// TIA Portal project "Phanloai_SP_height" (V16)
// Vorlageprojekt für das Buch mit Zielsystem S7-1200

(* hardware
DEVICE "S7-1200-Station_1"  S7-1200 Station
   slot 0: "Baugruppenträger_0"  Rack  V1.0
   slot 1: "PLC_1"  CPU 1211C DC/DC/DC  6ES7 211-1AE40-0XB0  V4.1
DEVICE "PC-System_1"  SIMATIC PC station
   slot 0: "SIMATIC PC station"  Rail  SIMATIC PC-Station  V1.0
      slot 125: "Stationmanager"  Station_Manager  V6.0.4
   slot 1: "HMI_RT_1"  WinCC RT Advanced  6AV2 104-0xxxx-xxxx  16.0.0.0
      slot 33792: "Computer interface"  Host interface
   slot 2: "IE general_1"  IE General  IE_CP  V8.2.0
*)

// ===== PLC "PLC_1"  CPU 1211C DC/DC/DC =====

VAR_GLOBAL   // PLC tag table "Standard-Variablentabelle"
   "M_Start" AT %M10.0 : Bool;
   "M_Stop" AT %M10.1 : Bool;
   "Den_M_Start" AT %M10.5 : Bool;
   "M_Pause" AT %M10.2 : Bool;
END_VAR

VAR_GLOBAL   // PLC tag table "INOUT"
   "START" AT %E0.0 : Bool;
   "STOP" AT %E0.1 : Bool;
   "Den START" AT %Q0.5 : Bool;
   "BT1" AT %A0.0 : Bool;
   "SS0" AT %I0.2 : Bool;
   "Pusher 0" AT %Q0.1 : Bool;
   "BT2" AT %Q0.4 : Bool;
   "PAUSE" AT %I0.5 : Bool;
   "SS1" AT %I0.3 : Bool;
   "Pusher 1" AT %Q0.2 : Bool;
   "Light 0" AT %Q1.0 : Bool;
   "Light 1" AT %Q1.1 : Bool;
   "Light 2" AT %Q1.2 : Bool;
   "Den STOP" AT %Q0.7 : Bool;
   "Den PAUSE" AT %Q0.6 : Bool;
   "SS2" AT %I0.4 : Bool;
END_VAR

VAR_GLOBAL   // PLC tag table "DEM_SP"
   "So SP vua" AT %QD34 : DWord;
   "So SP cao" AT %QD30 : DWord;
   "So SP thap" AT %QD38 : DWord;
END_VAR

VAR_GLOBAL   // PLC tag table "Temp_Vars"
   "P_Trig2" AT %M0.2 : Bool;
   "P_Trig3" AT %M0.4 : Bool;
   "P_Trig4" AT %M0.5 : Bool;
   "Temp1" AT %M0.6 : Bool;
   "P_Trig5" AT %M0.7 : Bool;
   "Temp" AT %M1.0 : Bool;
   "P_Trig1" AT %M1.1 : Bool;
   "Temp0" AT %M1.2 : Bool;
END_VAR

DATA_BLOCK "DB_VisualStudio"   // DB1
{ S7_Optimized_Access := 'TRUE' }
VERSION : 0.1
   VAR
      displayState : Bool;
   END_VAR
BEGIN
END_DATA_BLOCK

// folder: System blocks/Program resources

DATA_BLOCK "IEC_Counter_0_DB"   // DB2
{ S7_Optimized_Access := 'TRUE' }
AUTHOR : Simatic
FAMILY : IEC
NAME : CNTR
VERSION : 1.0
// stored: InstanceOfName IEC_COUNTER
"IEC_COUNTER"
BEGIN
END_DATA_BLOCK

DATA_BLOCK "IEC_Timer_0_DB_1"   // DB3
{ S7_Optimized_Access := 'TRUE' }
AUTHOR : Simatic
FAMILY : IEC
NAME : IEC_TMR
VERSION : 1.0
// stored: InstanceOfName IEC_TIMER
"IEC_TIMER"
BEGIN
END_DATA_BLOCK

DATA_BLOCK "IEC_Counter_0_DB1"   // DB4
{ S7_Optimized_Access := 'TRUE' }
AUTHOR : Simatic
FAMILY : IEC
NAME : CNTR
VERSION : 1.0
// stored: InstanceOfName IEC_COUNTER
"IEC_COUNTER"
BEGIN
END_DATA_BLOCK

DATA_BLOCK "IEC_Counter_0_DB2"   // DB5
{ S7_Optimized_Access := 'TRUE' }
AUTHOR : Simatic
FAMILY : IEC
NAME : CNTR
VERSION : 1.0
// stored: InstanceOfName IEC_COUNTER
"IEC_COUNTER"
BEGIN
END_DATA_BLOCK

DATA_BLOCK "IEC_Timer_0_DB_2"   // DB6
{ S7_Optimized_Access := 'TRUE' }
AUTHOR : Simatic
FAMILY : IEC
NAME : IEC_TMR
VERSION : 1.0
// stored: InstanceOfName IEC_TIMER
"IEC_TIMER"
BEGIN
END_DATA_BLOCK

DATA_BLOCK "IEC_Timer_0_DB_4"   // DB9
{ S7_Optimized_Access := 'TRUE' }
AUTHOR : Simatic
FAMILY : IEC
NAME : IEC_TMR
VERSION : 1.0
// stored: InstanceOfName IEC_TIMER
"IEC_TIMER"
BEGIN
END_DATA_BLOCK

DATA_BLOCK "IEC_Timer_0_DB_5"   // DB10
{ S7_Optimized_Access := 'TRUE' }
AUTHOR : Simatic
FAMILY : IEC
NAME : IEC_TMR
VERSION : 1.0
// stored: InstanceOfName IEC_TIMER
"IEC_TIMER"
BEGIN
END_DATA_BLOCK

// folder: (top level)

FUNCTION "MHJ-PLC-Lab-Function-S71200" : Void   // FC9000, SCL
{ S7_Optimized_Access := 'TRUE' }
VERSION : 0.1
   VAR_TEMP
      rdTimeReturn : Int;
      outputTime : DTL;
      SyncVal : Byte;
      forVal : Int;
      forVal_2 : Int;
      Value : Byte;
   END_VAR
   VAR CONSTANT
      CompVal : Byte := 16#34;
      Value_01 : Byte := 16#11;
      Value_01_DW : DWord := 16#A165_D992;
      Value_02_DW : DWord := 16#58BE_4401;
   END_VAR
BEGIN

   #Value:=PEEK(area := 16#82,
        dbNumber := 0,
        byteOffset := 511);
   #Value := #Value + 1;

   POKE(area := 16#82,
        dbNumber := 0,
        byteOffset := 511,
        value := #Value);

   POKE(area:=16#81,
        dbNumber:=0,
        byteOffset:=1016,
        value:=#Value_01_DW);
   POKE(area := 16#81,
        dbNumber := 0,
        byteOffset := 1020,
        value := #Value_02_DW);

   POKE(area := 16#81,
        dbNumber := 0,
        byteOffset := 511,
        value := B#16#00);

   FOR #forVal := 0 TO 120 DO
       FOR #forVal_2:=0 TO 10 DO
           #rdTimeReturn:=RD_SYS_T(#outputTime);
           #rdTimeReturn := WR_SYS_T(#outputTime);
           #rdTimeReturn := RD_SYS_T(#outputTime);
           #rdTimeReturn := WR_SYS_T(#outputTime);
       END_FOR;
       #SyncVal:= PEEK(area := 16#81,
                      dbNumber := 0,
                      byteOffset := 511);
       IF #SyncVal = #CompVal THEN
          GOTO M_1;
       END_IF;
   END_FOR;
   RETURN;

   M_1:
   POKE(area := 16#81,
        dbNumber := 0,
        byteOffset := 511,
        value := B#16#0);
END_FUNCTION

ORGANIZATION_BLOCK "Main"   // OB1, LAD, ProgramCycle
TITLE = "Main Program Sweep (Cycle)"
{ S7_Optimized_Access := 'TRUE' }
VERSION : 0.1
   VAR_INPUT
      Initial_Call : Bool;   // Initial call of this OB
      Remanence : Bool;   // =True, if remanent data are available
   END_VAR
   VAR_TEMP   // added for the SCL form of the ladder/FBD networks
      _w1 : Bool;
   END_VAR
BEGIN

REGION Network 1: Konnektierungsbaustein für PLC-Lab
   // Im Netzwerk 1 wird der Konnektierungsbaustein für PLC-Lab aufgerufen.
   // Dieser Aufruf darf nicht entfernt werden!
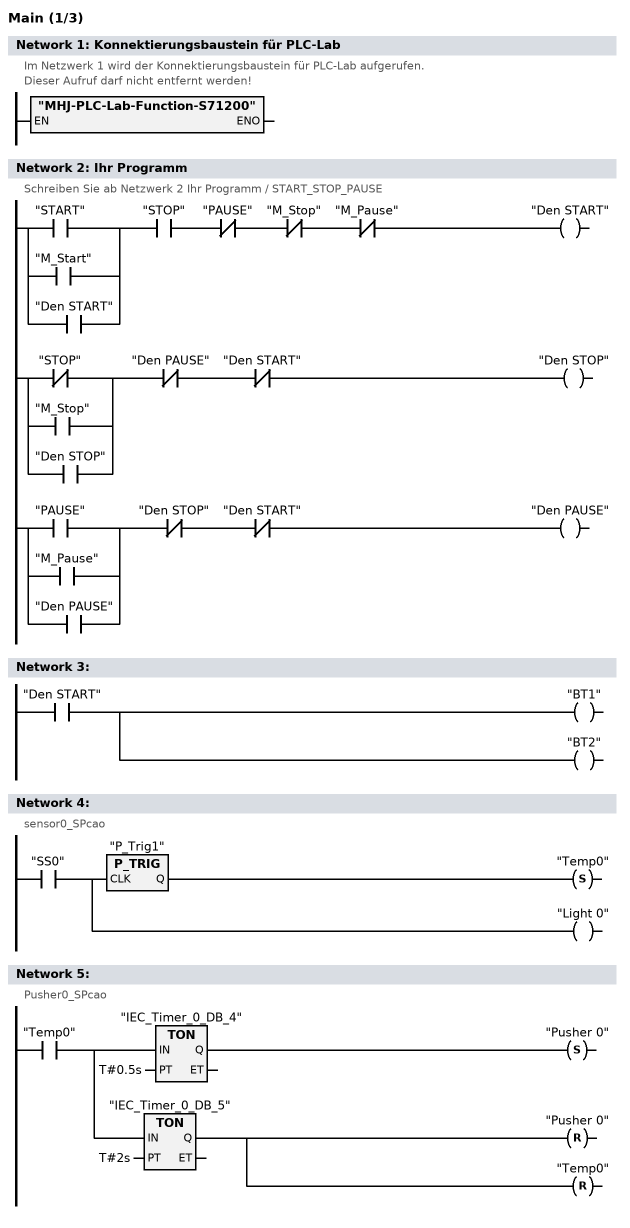
   RUNG wire#powerrail
      "MHJ-PLC-Lab-Function-S71200"()
   END_RUNG
   // the same network as SCL:
   "MHJ-PLC-Lab-Function-S71200"();
END_REGION

REGION Network 2: Ihr Programm
   // Schreiben Sie ab Netzwerk 2 Ihr Programm / START_STOP_PAUSE
   RUNG wire#powerrail
      Contact( "START" )
      wire#w1
      Contact( "STOP" )
      I_Contact( "PAUSE" )
      I_Contact( "M_Stop" )
      I_Contact( "M_Pause" )
      Coil( "Den START" )
   END_RUNG
   RUNG wire#powerrail
      Contact( "M_Start" )
   END_RUNG wire#w1
   RUNG wire#powerrail
      Contact( "Den START" )
   END_RUNG wire#w1
   RUNG wire#powerrail
      I_Contact( "STOP" )
      wire#w2
      I_Contact( "Den PAUSE" )
      I_Contact( "Den START" )
      Coil( "Den STOP" )
   END_RUNG
   RUNG wire#powerrail
      Contact( "M_Stop" )
   END_RUNG wire#w2
   RUNG wire#powerrail
      Contact( "Den STOP" )
   END_RUNG wire#w2
   RUNG wire#powerrail
      Contact( "PAUSE" )
      wire#w3
      I_Contact( "Den STOP" )
      I_Contact( "Den START" )
      Coil( "Den PAUSE" )
   END_RUNG
   RUNG wire#powerrail
      Contact( "M_Pause" )
   END_RUNG wire#w3
   RUNG wire#powerrail
      Contact( "Den PAUSE" )
   END_RUNG wire#w3
   // the same network as SCL:
   "Den START" := ("START" OR "M_Start" OR "Den START") AND "STOP" AND NOT "PAUSE" AND NOT "M_Stop" AND NOT "M_Pause";
   "Den STOP" := (NOT "STOP" OR "M_Stop" OR "Den STOP") AND NOT "Den PAUSE" AND NOT "Den START";
   "Den PAUSE" := ("PAUSE" OR "M_Pause" OR "Den PAUSE") AND NOT "Den STOP" AND NOT "Den START";
END_REGION

REGION Network 3
   RUNG wire#powerrail
      Contact( "Den START" )
      wire#w1
      Coil( "BT1" )
   END_RUNG
   RUNG wire#w1
      Coil( "BT2" )
   END_RUNG
   // the same network as SCL:
   "BT1" := "Den START";
   "BT2" := "Den START";
END_REGION

REGION Network 4
   // sensor0_SPcao
   RUNG wire#powerrail
      Contact( "SS0" )
      wire#w1
      P_Trig( "P_Trig1" )
      S_Coil( "Temp0" )
   END_RUNG
   RUNG wire#w1
      Coil( "Light 0" )
   END_RUNG
   // the same network as SCL:
   #_w1 := "SS0" AND NOT "P_Trig1";   // rising edge
   "P_Trig1" := "SS0";
   IF #_w1 THEN "Temp0" := TRUE; END_IF;
   "Light 0" := "SS0";
END_REGION

REGION Network 5
   // Pusher0_SPcao
   "IEC_Timer_0_DB_4".TON(IN := "Temp0", PT := T#0.5s);
   IF "IEC_Timer_0_DB_4".Q THEN "Pusher 0" := TRUE; END_IF;
   "IEC_Timer_0_DB_5".TON(IN := "Temp0", PT := T#2s);
   IF "IEC_Timer_0_DB_5".Q THEN
       "Pusher 0" := FALSE;
       "Temp0" := FALSE;
   END_IF;
END_REGION

REGION Network 6
   // Dem SP cao
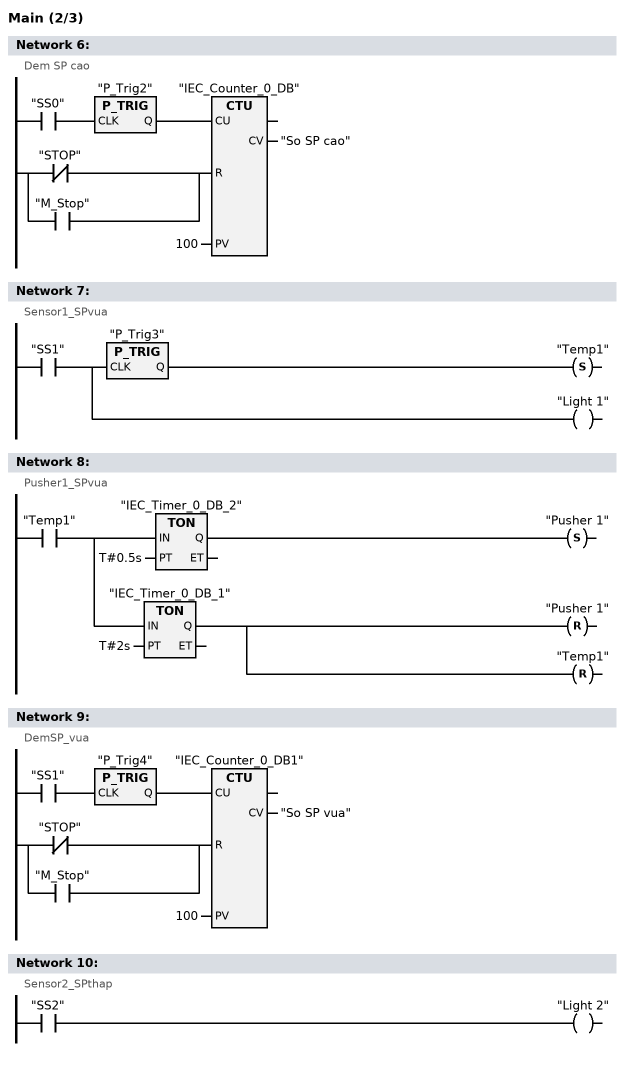
   #_w1 := "SS0" AND NOT "P_Trig2";   // rising edge
   "P_Trig2" := "SS0";
   "IEC_Counter_0_DB".CTU(CU := #_w1, R := NOT "STOP" OR "M_Stop", PV := 100, CV => "So SP cao");
END_REGION

REGION Network 7
   // Sensor1_SPvua
   RUNG wire#powerrail
      Contact( "SS1" )
      wire#w1
      P_Trig( "P_Trig3" )
      S_Coil( "Temp1" )
   END_RUNG
   RUNG wire#w1
      Coil( "Light 1" )
   END_RUNG
   // the same network as SCL:
   #_w1 := "SS1" AND NOT "P_Trig3";   // rising edge
   "P_Trig3" := "SS1";
   IF #_w1 THEN "Temp1" := TRUE; END_IF;
   "Light 1" := "SS1";
END_REGION

REGION Network 8
   // Pusher1_SPvua
   "IEC_Timer_0_DB_2".TON(IN := "Temp1", PT := T#0.5s);
   IF "IEC_Timer_0_DB_2".Q THEN "Pusher 1" := TRUE; END_IF;
   "IEC_Timer_0_DB_1".TON(IN := "Temp1", PT := T#2s);
   IF "IEC_Timer_0_DB_1".Q THEN
       "Pusher 1" := FALSE;
       "Temp1" := FALSE;
   END_IF;
END_REGION

REGION Network 9
   // DemSP_vua
   #_w1 := "SS1" AND NOT "P_Trig4";   // rising edge
   "P_Trig4" := "SS1";
   "IEC_Counter_0_DB1".CTU(CU := #_w1, R := NOT "STOP" OR "M_Stop", PV := 100, CV => "So SP vua");
END_REGION

REGION Network 10
   // Sensor2_SPthap
   RUNG wire#powerrail
      Contact( "SS2" )
      Coil( "Light 2" )
   END_RUNG
   // the same network as SCL:
   "Light 2" := "SS2";
END_REGION

REGION Network 11
   // Dem SP thap
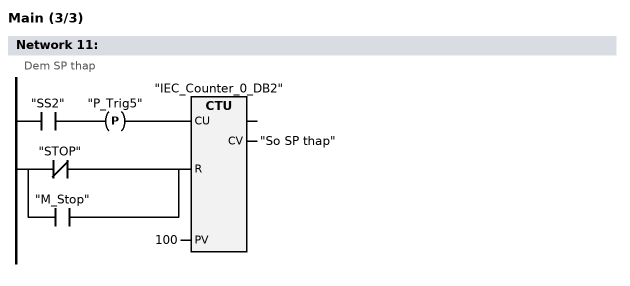
   #_w1 := "SS2" AND NOT "P_Trig5";   // rising edge
   "P_Trig5" := "SS2";
   "IEC_Counter_0_DB2".CTU(CU := #_w1, R := NOT "STOP" OR "M_Stop", PV := 100, CV => "So SP thap");
END_REGION
END_ORGANIZATION_BLOCK

(* ===== HMI "HMI_RT_1" =====
system functions are stored by id; their names below are inferred from use
connection "HMI_Connection_1": ETHERNET, S7_1200_OMS

HMI tags "Default tag table"
   "START" : Bool = PLC START AT %I0.0, 1 s
   "STOP" : Bool = PLC STOP AT %I0.1, 1 s
   "DUNG" : Bool = PLC PAUSE AT %I0.5, 1 s
   "LED" : Bool = PLC "Den START" AT %Q0.5, 1 s
   "Den STOP" : Bool = PLC "Den STOP" AT %Q0.7, 1 s
   "Den DUNG" : Bool = PLC "Den PAUSE" AT %Q0.6, 1 s
   "Light 1" : Bool = PLC "Light 0" AT %Q1.0, 1 s
   "Light 2" : Bool = PLC "Light 1" AT %Q1.1, 1 s
   "Light 3" : Bool = PLC "Light 2" AT %Q1.2, 1 s
   "So SP cao" : DWord = PLC "So SP cao" AT %QD30, 1 s
   "So SP vua" : DWord = PLC "So SP vua" AT %QD34, 1 s
   "So SP thap" : DWord = PLC "So SP thap" AT %QD38, 1 s

screen "Screen_1" 800x600
   TextField "Text field_1" at 53,99 size 627x48; Text 'PHAN LOAI SP THEO CHIEU CAO'
   Button "Button_1" at 49,206 size 119x48; TextOff 'START'
      on Release: ResetBit("START")
      on Press: SetBit("START")
   Button "Button_2" at 49,274 size 119x48; TextOff 'STOP'
      on Release: ResetBit("STOP")
      on Press: SetBit("STOP")
   Button "Button_3" at 48,352 size 119x48; TextOff 'PAUSE'
      on Release: ResetBit("DUNG")
      on Press: SetBit("DUNG")
   Circle "Circle_1" at 187,207 size 48x48
      Appearance <- "LED"
   Circle "Circle_2" at 187,275 size 48x48
      Appearance <- "Den STOP"
   Circle "Circle_3" at 187,352 size 48x48
      Appearance <- "Den DUNG"
   Circle "Circle_4" at 303,428 size 48x48
      Appearance <- "Light 1"
   Circle "Circle_5" at 443,428 size 48x48
      Appearance <- "Light 2"
   Circle "Circle_6" at 591,425 size 48x48
      Appearance <- "Light 3"
   TextField "Text field_2" at 271,384 size 109x38; Text 'Light 1'
   TextField "Text field_3" at 421,378 size 83x45; Text 'Light 2'
   TextField "Text field_4" at 565,382 size 100x39; Text 'Light 3'
   TextField "Text field_5" at 281,287 size 87x30; Text 'CAO'
   TextField "Text field_6" at 436,291 size 76x22; Text 'VUA'
   TextField "Text field_7" at 570,290 size 107x22; Text 'THAP'
   IOField "I/O field_1" at 280,317 size 96x32; FormatPattern 999
      ProcessValue <- "So SP cao"
   IOField "I/O field_2" at 424,318 size 96x32; FormatPattern 999
      ProcessValue <- "So SP vua"
   IOField "I/O field_3" at 575,316 size 96x32; FormatPattern 999
      ProcessValue <- "So SP thap"
*)